{attribute 'qualified_only'}
{attribute 'to_string'}
TYPE E_FaultTypes : // Fault types, sorted by severity
(
	OM, // Operator message
	OW, // Operator warning
	MC, // Missing condition
	CF, // Cycle Fault
	FF, // Fatal fault
	_ENUM_SIZE // Always the last item in the enumerator
) UINT;
END_TYPE

(* stored: Version 1.1.0.1, ProductVersion 3.1.4024.11
   EnumerationTextList E_FaultTypes: Id {80d266b1-3eb3-4c6d-b0bb-2f4400a81ab3} *)
